Omron CX-Programmer project NewProject (CX-Programmer 9.81)

# PLC Lateh: CJ1M CPU11

## Program NewProgram1 (cyclic task 0)
Local symbols
BE 0.00 BOOL  ; Botão emergência
BS 0.01 BOOL  ; Botâo STOP
B_Start 0.02 BOOL  ; Botâo start
NO 0.04 BOOL  ; Normalmente aberto
R1 0.03 BOOL  ; Relé 1
RA1 0.05 BOOL  ; Bobine 1

### Section Section1

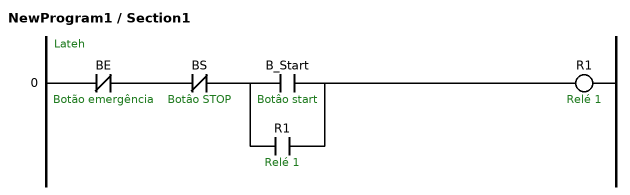
; rung 0: Lateh
LDNOT BE  ; Botão emergência
ANDNOT BS  ; Botâo STOP
LD B_Start  ; Botâo start
OR R1  ; Relé 1
ANDLD
OUT R1  ; Relé 1

### Section END
; rung 0
END(001)